// TIA Portal V17 export
// export: Created 2022-07-20T06:59:39.0020974Z, ExportSetting WithDefaults, DisplayName Totally Integrated Automation Portal, DisplayVersion V17, DisplayName TIA Portal Openness, DisplayVersion V17, DisplayName TIA Portal Version Control Interface, DisplayVersion V17, DisplayName SINAMICS Startdrive Advanced, DisplayVersion V17, DisplayName SINAMICS Startdrive G130, G150, S120, S150, SINAMICS MV, S210, DisplayVersion V17, DisplayName SINAMICS Startdrive G110M, G120, G120C, G120D, G120P, G115D, DisplayVersion V17, DisplayName STEP 7 Professional, DisplayVersion V17, DisplayName STEP 7 Safety, DisplayVersion V17, DisplayName WinCC Advanced, DisplayVersion V17
FUNCTION "FC10010_ScalingPercentageToAnalog" : Void   // FC10010, LAD
TITLE = FC10010_ScalingPercentageToAnalog
{ S7_Optimized_Access := 'TRUE' }
AUTHOR : Jonathan
FAMILY : 1001x_CONVERT
VERSION : 1.0
// Release note : 
// 1.0 - Feature developped
// stored: AutoNumber false, IsIECCheckEnabled false, SetENOAutomatically false, UDAEnableTagReadback false
   VAR_INPUT
      SetPoint : Real;
   END_VAR
   VAR_OUTPUT
      AnalogValue : Int;
   END_VAR
   VAR_TEMP
      SetPointNorm : Real;
   END_VAR
BEGIN

REGION Network 1: Normalize the set point
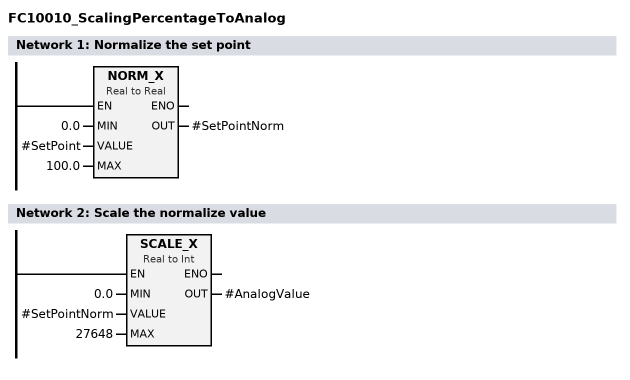
   RUNG wire#powerrail
      { S7_Templates := "[SrcType := Real, DestType := Real]" } Normalize(min := 0.0, value := #SetPoint, max := 100.0, out => #SetPointNorm)
   END_RUNG
   // the same network as SCL:
   #SetPointNorm := NORM_X(MIN := 0.0, VALUE := #SetPoint, MAX := 100.0);
END_REGION

REGION Network 2: Scale the normalize value
   RUNG wire#powerrail
      { S7_Templates := "[SrcType := Real, DestType := Int]" } Scale(min := 0.0, value := #SetPointNorm, max := 27648, out => #AnalogValue)
   END_RUNG
   // the same network as SCL:
   #AnalogValue := SCALE_X(MIN := 0.0, VALUE := #SetPointNorm, MAX := 27648);
END_REGION
END_FUNCTION
